Staubli VAL3: Day6.pjx

--- Day6.pjx ---
Parameters version=s8.13.1Cs9_BS2800 stackSize=5000 millimeterUnit=true
Program file=generation_generator.pgx
Program file=start.pgx
Program file=stop.pgx
Data file=Day6.dtx
Library alias=util path=Disk://helpers/helpers.pjx
Library alias=math path=Disk://math/math.pjx
Library alias=str path=Disk://string/string.pjx
Type name=lists path=Disk://types/lists/lists.pjx
Type name=lists_num path=Disk://types/lists_num/lists_num.pjx

--- Day6.dtx ---
string sInput
num nInput
lists lResult
  [0]
    string sString
num nResult
num nInput2
num nCounter[9]

--- start.pgx ---
program start()
begin

  // read file
  call util:readFile("Disk://input_day6.txt", sInput)
  // sInput[0] = "905,103 -> 905,82"

  call str:splitString(sInput,",", lResult)

  call util:vec2num(lResult.sString, nInput)
  call util:vec2num(lResult[1].sString, nInput2)

  call util:mergeVectors(nInput,nInput2, nResult)
  call util:vec2num(lResult[2].sString, nInput2)
  call util:mergeVectors(nResult,nInput2, nInput)

  // PUZZLE 1
  call generation_generator(80)
  // 361169

  // PUZZLE 2
  call generation_generator(256)
  // 1634946868992

end

--- generation_generator.pgx ---
program generation_generator(num x_nDays)
  local num l_nElement
  local num l_nValue
  local num l_nDays
  local num l_nNewFishes
  local num l_nRESULT
begin

  // count values
  resize(nCounter,1,1)
  nCounter = 0
  resize(nCounter,1,9)
  for l_nElement = 0 to size(nInput)-1
    for l_nValue = 0 to 8
      if nInput[l_nElement] == l_nValue
        nCounter[l_nValue] = nCounter[l_nValue] + 1
      endIf
    endFor
  endFor

  for l_nDays = 1 to x_nDays
    l_nNewFishes = nCounter[0]

    delete(nCounter[0])

    nCounter[6] = nCounter[6] + l_nNewFishes
    append(nCounter)
    nCounter[8] = l_nNewFishes
  endFor

  call math:sum(nCounter, l_nRESULT)
  call util:printNum(l_nRESULT)


end
